FUNCTION_BLOCK StartProgramTask EXTENDS TcoCore.TcoTask 
VAR

	_stopType: TcoAbstractions.eTcoRoboticsStopType;
END_VAR
VAR
    {attribute 'hide'} 
	_progress : INT := 0;
    {attribute 'hide'} 
	_infoTimer :  TON;
    {attribute 'hide'} 
	_errorTimer :  TON;
    {attribute 'hide'} 
	_varInfo : __SYSTEM.VAR_INFO;
    {attribute 'hide'} 
	_sb : TcoCore.StringBuilder;
	{attribute 'hide'}
	_blink:TcoUtilities.TcoBlinker(THIS^);
END_VAR

VAR_IN_OUT
    inoConfig 	: TcoIrc5_Config_v_1_x_x;
	inoControl 	: TcoIrc5_Control_v_1_x_x;
	inoStatus 	: TcoIrc5_Status_v_1_x_x;	
END_VAR



IF Execute() THEN
	_blink(inOnTime:=T#500MS,inOffTime:=T#500MS);

	IF _progress = 0 THEN
		IF NOT __ISVALIDREF(inoControl) THEN
			_varInfo :=__VARINFO(inoControl);
			Messenger.Programming(_sb.Clear().Append('<#Invalid reference: #>').Append(_varInfo.Symbol).ToString()).Pin();
		ELSIF NOT __ISVALIDREF(inoConfig) THEN                                                  
			_varInfo :=__VARINFO(inoConfig);                                                    
			Messenger.Programming(_sb.Clear().Append('<#Invalid reference: #>').Append(_varInfo.Symbol).ToString()).Pin();
		ELSIF NOT __ISVALIDREF(inoStatus) THEN                                                  
			_varInfo :=__VARINFO(inoStatus);                                                    
			Messenger.Programming(_sb.Clear().Append('<#Invalid reference: #>').Append(_varInfo.Symbol).ToString()).Pin();
			ELSE
			_progress := _progress + 1;
		END_IF

	END_IF
	IF _progress = 1 THEN
		inoControl.StartProgram:=_blink.outQ;
		
		IF  inoStatus.State.CycleOn AND NOT inoStatus.State.SystemInputBusy THEN
				inoControl.StartProgram:=FALSE;
		END_IF
	END_IF;		
	
	

    DoneWhen(inoStatus.State.CycleOn AND NOT inoStatus.State.SystemInputBusy);
    CallTimers(TRUE);
	
	THIS^.ThrowWhen(_errorTimer.Q);
END_IF

METHOD CallTimers
VAR_INPUT
	inValue : BOOL;
END_VAR
IF  __ISVALIDREF(inoConfig) THEN  
_infoTimer(IN := inValue, PT := THIS^.inoConfig.InfoTime);
_errorTimer(IN := inValue, PT := THIS^.inoConfig.ErrorTime);
END_IF;
END_METHOD

METHOD PUBLIC FB_init : BOOL
VAR_INPUT
    bInitRetains : BOOL; // if TRUE, the retain variables are initialized (warm start / cold start)
    bInCopyCode : BOOL; // if TRUE, the instance afterwards gets moved into the copy code (online change)
  	ParentObject : ITcoObject;	
END_VAR
END_METHOD

METHOD INTERNAL InvokeWithParams : ITcoTaskStatus
VAR_INPUT
	inStopType : eTcoRoboticsStopType;
END_VAR
_stopType := inStopType;
InvokeWithParams := THIS^.Invoke();
END_METHOD

(*~
	<docu>
		<summary>
			Executes when task is aborted.
		</summary>			
	</docu>	
~*)
METHOD PROTECTED OnAbort
IF  __ISVALIDREF(inoStatus) THEN   THIS^.inoStatus.ActionDescription := '<#Stop program was aborted, while not yet completed!#>';END_IF;
END_METHOD

(*~
	<docu>
		<summary>
			Executes when task reaches the ```Done``` state .
		</summary>			
	</docu>	
~*)
METHOD PROTECTED OnDone
IF  __ISVALIDREF(inoStatus) THEN  THIS^.inoStatus.ActionDescription := '<#Stop program was completed successfully.#>';END_IF; 
_progress:=0;
END_METHOD

(*~
	<docu>
		<summary>
			Executes when task reaches the ```Error``` state.
			<para>
				Do not confuse with <see cref="PlcDocu.TcoCore.TcoTask.WhileError()"/>, that is called cyclically until '''Error''' state is left.
			</para>
		</summary>			
	</docu>	
~*)
METHOD PROTECTED OnError
IF  __ISVALIDREF(inoStatus) THEN   THIS^.inoStatus.ActionDescription := '<#Stopping program with error.#>'; END_IF;
END_METHOD

METHOD PROTECTED OnStart
IF  __ISVALIDREF(inoStatus) THEN  THIS^.inoStatus.ActionDescription := '<#Stopping program started.#>'; END_IF; 
CallTimers(FALSE);
END_METHOD

(*~
	<docu>
		<summary>
			Restores this instance to the Ready state. Can be called explicitly or from within one of the restore mechanisms.
			<para>
				See also <see cref="PlcDocu.TcoCore.TcoTask.AutoRestorable()"/>
			</para>
		</summary>			
	</docu>	
~*)
METHOD Restore : ITcoRestorable
SUPER^.Restore();
_progress := 0;
CallTimers(FALSE);
Messenger.UnPin();
END_METHOD

END_FUNCTION_BLOCK

(* stored: Version 1.1.0.1, ProductVersion 3.1.4024.12
   POU StartProgramTask: Id {c63fdbca-73e5-04fc-22b5-7387f2d6f967}, SpecialFunc None
   Method CallTimers: Id {e8b8b07f-fae4-02be-1033-9572e3c33402}
   Method FB_init: Id {78852108-bba5-089f-1a26-a6bd957eb025}
   Method InvokeWithParams: Id {795a573d-7973-0c5f-3c9a-d3a35252b0a6}
   Method OnAbort: Id {1904980f-061a-047e-2687-a3a2361e384a}
   Method OnDone: Id {b2efc703-d968-044f-056d-8a5cb67c88f1}
   Method OnError: Id {ce609b33-6a6d-09d3-27e1-dc4f64dd8efc}
   Method OnStart: Id {37f34ec0-7926-0f27-366f-58ec49562eab}
   Method Restore: Id {98fadc18-5956-0e3d-0700-a1266e3d180e} *)
